// TIA Portal V20 export
DATA_BLOCK "LBP_Axis17"   // DB47
TITLE = Axis-specific signals / Signaux spécifiques à un axe
{ S7_Optimized_Access := 'FALSE' }
AUTHOR : SINUMERIK
FAMILY : SINUMERIK_ONE
VERSION : 6.24
// Interface between user program and axis/spindle, contains signals from/to axis/spindle 17 / Interface entre programme utilisateur et axe/broche, contient des signaux de/vers axe/broche 17
// stored: AutoNumber false, InstanceOfName LBP_typeAxisX, InstanceOfType UDT
"LBP_typeAxisX"
   // VAR RETAIN
   //    A_FD_OR : Byte;
   //    A_DriveEnable : Bool;
   //    A_AckFixedStop : Bool;
   //    A_SensorFixedStop : Bool;
   //    A_ASpDisable : Bool;
   //    A_Follow_upMode : Bool;
   //    A_PosMeas1 : Bool;
   //    A_PosMeas2 : Bool;
   //    A_ORactive : Bool;
   //    A_SWCam : Bool;
   //    A_ContrEnable : Bool;
   //    A_DelDTGSpReset : Bool;
   //    A_Clamp : Bool;
   //    A_RefVal1 : Bool;
   //    A_RefVal2 : Bool;
   //    A_RefVal3 : Bool;
   //    A_RefVal4 : Bool;
   //    A_ExtZO : Bool;
   //    A_EnabTravFixedStop : Bool;
   //    A_FixedFD1 : Bool;
   //    A_FixedFD2 : Bool;
   //    A_FixedFD3 : Bool;
   //    A_FixedFD4 : Bool;
   //    A_VelocSpeedLimit : Bool;
   //    A_PrgtestAxRel : Bool;
   //    A_HW1 : Bool;
   //    A_HW2 : Bool;
   //    A_HW3 : Bool;
   //    A_FDSpStop : Bool;
   //    A_Disable : Bool;
   //    A_RapidTrOR : Bool;
   //    A_Minus : Bool;
   //    A_Plus : Bool;
   //    A_INC1 : Bool;
   //    A_INC10 : Bool;
   //    A_INC100 : Bool;
   //    A_INC1000 : Bool;
   //    A_INC10000 : Bool;
   //    A_INCVar : Bool;
   //    A_ContManTravel : Bool;
   //    f5_7 : Bool;
   //    A_OEMAxis : Byte;
   //    A_InvHWDirOfRot : Bool;
   //    f7_1 : Bool;
   //    f7_2 : Bool;
   //    f7_3 : Bool;
   //    f7_4 : Bool;
   //    f7_5 : Bool;
   //    f7_6 : Bool;
   //    f7_7 : Bool;
   //    A_NCASpChanA : Bool;
   //    A_NCASpChanB : Bool;
   //    A_NCASpChanC : Bool;
   //    A_NCASpChanD : Bool;
   //    A_NCASpStrobe : Bool;
   //    f8_5 : Bool;
   //    f8_6 : Bool;
   //    A_PLCASp : Bool;
   //    A_Para_A : Bool;
   //    A_Para_B : Bool;
   //    A_Para_C : Bool;
   //    A_LockParSetDef : Bool;
   //    f9_4 : Bool;
   //    f9_5 : Bool;
   //    f9_6 : Bool;
   //    f9_7 : Bool;
   //    A_REPOSDelay : Bool;
   //    f10_1 : Bool;
   //    f10_2 : Bool;
   //    f10_3 : Bool;
   //    f10_4 : Bool;
   //    f10_5 : Bool;
   //    f10_6 : Bool;
   //    f10_7 : Bool;
   //    A_StartBrakeTest : Bool;
   //    f11_1 : Bool;
   //    f11_2 : Bool;
   //    f11_3 : Bool;
   //    f11_4 : Bool;
   //    f11_5 : Bool;
   //    f11_6 : Bool;
   //    f11_7 : Bool;
   //    A_HWLimitMinus : Bool;
   //    A_HWLimitPlus : Bool;
   //    A_SWLimit2Minus : Bool;
   //    A_SWLimit2Plus : Bool;
   //    A_ModuloLimitEn : Bool;
   //    f12_5 : Bool;
   //    f12_6 : Bool;
   //    A_DelayRef : Bool;
   //    A_JogFixPPos0 : Bool;
   //    A_JogFixPPos1 : Bool;
   //    A_JogFixPPos2 : Bool;
   //    A_JogToPos : Bool;
   //    f13_4 : Bool;
   //    f13_5 : Bool;
   //    f13_6 : Bool;
   //    f13_7 : Bool;
   //    A_ProgtestSuppress : Bool;
   //    A_ProgtestActivate : Bool;
   //    f14_2 : Bool;
   //    f14_3 : Bool;
   //    f14_4 : Bool;
   //    f14_5 : Bool;
   //    f14_6 : Bool;
   //    f14_7 : Bool;
   //    f15 : Byte;
   //    A_ActGearA : Bool;
   //    A_ActGearB : Bool;
   //    A_ActGearC : Bool;
   //    A_GearChangeOv : Bool;
   //    A_Sp1Syn : Bool;
   //    A_Sp2Syn : Bool;
   //    A_NoMonitorGear : Bool;
   //    A_DeleteS : Bool;
   //    A_FD_ORSp : Bool;
   //    f17_1 : Bool;
   //    f17_2 : Bool;
   //    f17_3 : Bool;
   //    A_Sp1SynP : Bool;
   //    A_Sp2SynP : Bool;
   //    A_M3M4Inv : Bool;
   //    f17_7 : Bool;
   //    f18_0 : Bool;
   //    f18_1 : Bool;
   //    f18_2 : Bool;
   //    f18_3 : Bool;
   //    A_OscilPLC : Bool;
   //    A_OscilSpeed : Bool;
   //    A_SetRotDirectRight : Bool;
   //    A_SetRotDirectLeft : Bool;
   //    A_SpOR : Byte;
   //    f20_0 : Bool;
   //    A_RUEncQuStop : Bool;
   //    f20_2 : Bool;
   //    A_SpeedSetpSmooth : Bool;
   //    f20_4 : Bool;
   //    A_HoldBrakeToOpen : Bool;
   //    f20_6 : Bool;
   //    f20_7 : Bool;
   //    A_ParA : Bool;
   //    A_ParB : Bool;
   //    A_ParC : Bool;
   //    A_MotA : Bool;
   //    A_MotB : Bool;
   //    A_MotOK : Bool;
   //    A_IntegratDisable : Bool;
   //    A_PulseEnable : Bool;
   //    f22_0 : Bool;
   //    f22_1 : Bool;
   //    f22_2 : Bool;
   //    f22_3 : Bool;
   //    f22_4 : Bool;
   //    f22_5 : Bool;
   //    f22_6 : Bool;
   //    f22_7 : Bool;
   //    f23_0 : Bool;
   //    f23_1 : Bool;
   //    f23_2 : Bool;
   //    f23_3 : Bool;
   //    f23_4 : Bool;
   //    f23_5 : Bool;
   //    f23_6 : Bool;
   //    f23_7 : Bool;
   //    f24_0 : Bool;
   //    A_ControlAx : Bool;
   //    f24_2 : Bool;
   //    f24_3 : Bool;
   //    A_TorqComp : Bool;
   //    A_ChangSetpOutAss0 : Bool;
   //    A_ChangSetpOutAss1 : Bool;
   //    A_MS : Bool;
   //    A_DynBComp : Bool;
   //    f25_1 : Bool;
   //    f25_2 : Bool;
   //    f25_3 : Bool;
   //    f25_4 : Bool;
   //    f25_5 : Bool;
   //    f25_6 : Bool;
   //    f25_7 : Bool;
   //    f26_0 : Bool;
   //    f26_1 : Bool;
   //    f26_2 : Bool;
   //    A_CompContr : Bool;
   //    A_FollowAxOv : Bool;
   //    f26_5 : Bool;
   //    f26_6 : Bool;
   //    f26_7 : Bool;
   //    A_DEPMCS : Bool;
   //    A_DEPBCS : Bool;
   //    A_Corr : Bool;
   //    A_HIAxMove : Bool;
   //    A_StopDEPMCS : Bool;
   //    A_StopDEPBCS : Bool;
   //    A_StopCorr : Bool;
   //    A_StopHIAxMove : Bool;
   //    A_OscillAxExtRev : Bool;
   //    A_AxReset : Bool;
   //    A_AxResume : Bool;
   //    A_SetRP : Bool;
   //    A_ChangeRP : Bool;
   //    A_StopRP : Bool;
   //    A_Stop : Bool;
   //    A_PLCAxis : Bool;
   //    f29_0 : Bool;
   //    f29_1 : Bool;
   //    f29_2 : Bool;
   //    f29_3 : Bool;
   //    A_StartGantSynRun : Bool;
   //    A_NoAutoSync : Bool;
   //    f29_6 : Bool;
   //    f29_7 : Bool;
   //    A_StopSpindle : Bool;
   //    A_StartCW : Bool;
   //    A_StartCCW : Bool;
   //    A_AutoGearStep : Bool;
   //    A_PosSpindle : Bool;
   //    f30_5 : Bool;
   //    f30_6 : Bool;
   //    f30_7 : Bool;
   //    f31_0 : Bool;
   //    f31_1 : Bool;
   //    f31_2 : Bool;
   //    f31_3 : Bool;
   //    A_Resynchronize : Bool;
   //    A_DisSync : Bool;
   //    A_Tracksync : Bool;
   //    A_DelSyncRunCorr : Bool;
   //    f32_0 : Bool;
   //    f32_1 : Bool;
   //    f32_2 : Bool;
   //    f32_3 : Bool;
   //    f32_4 : Bool;
   //    f32_5 : Bool;
   //    f32_6 : Bool;
   //    f32_7 : Bool;
   //    f33_0 : Bool;
   //    f33_1 : Bool;
   //    f33_2 : Bool;
   //    f33_3 : Bool;
   //    f33_4 : Bool;
   //    f33_5 : Bool;
   //    f33_6 : Bool;
   //    f33_7 : Bool;
   //    A_SI_SetpLimBit0 : Bool;
   //    A_SI_SetpLimBit1 : Bool;
   //    f34_2 : Bool;
   //    A_ActivateBrakeRampForSs2e : Bool;
   //    f34_4 : Bool;
   //    f34_5 : Bool;
   //    f34_6 : Bool;
   //    f34_7 : Bool;
   //    f35 : Byte;
   //    f36 : Array[36..55] of Byte;
   //    A_FeedDriveCAxEng : Bool;
   //    A_SpSpeedDisp : Bool;
   //    A_SpInsideClamp : Bool;
   //    f56_3 : Bool;
   //    f56_4 : Bool;
   //    f56_5 : Bool;
   //    f56_6 : Bool;
   //    f56_7 : Bool;
   //    f57 : Byte;
   //    f58 : Word;
   //    E_SpNA : Bool;
   //    E_NCU_Link : Bool;
   //    E_EncodFreq1 : Bool;
   //    E_EncodFreq2 : Bool;
   //    E_RefSyn1 : Bool;
   //    E_RefSyn2 : Bool;
   //    E_ExactCoarse : Bool;
   //    E_ExactFine : Bool;
   //    E_TravRequ : Bool;
   //    E_AxialAlarm : Bool;
   //    E_AxisReady : Bool;
   //    E_Follow_upMode : Bool;
   //    E_Stat : Bool;
   //    E_PositContr : Bool;
   //    E_SpeedContr : Bool;
   //    E_CurrentContr : Bool;
   //    E_SWCam : Bool;
   //    E_HWOverlay : Bool;
   //    E_RevFD : Bool;
   //    E_MeasAct : Bool;
   //    E_ActTravFStop : Bool;
   //    E_FixedStop : Bool;
   //    E_ForceFixedStop : Bool;
   //    E_AxContainerRot : Bool;
   //    E_AxReset : Bool;
   //    E_PLCCtrlAx : Bool;
   //    E_AxStop : Bool;
   //    E_AxSpDisable : Bool;
   //    E_StopDEPMCS : Bool;
   //    E_StopDEPBCS : Bool;
   //    E_StopCorr : Bool;
   //    E_StopHIAxMove : Bool;
   //    E_HW1 : Bool;
   //    E_HW2 : Bool;
   //    E_HW3 : Bool;
   //    f64_3 : Bool;
   //    E_TReqMinus : Bool;
   //    E_TReqPlus : Bool;
   //    E_TCMinus : Bool;
   //    E_TCPlus : Bool;
   //    E_INC1 : Bool;
   //    E_INC10 : Bool;
   //    E_INC100 : Bool;
   //    E_INC1000 : Bool;
   //    E_INC10000 : Bool;
   //    E_INCVar : Bool;
   //    E_ContManTravelAct : Bool;
   //    f65_7 : Bool;
   //    E_OEMAxis : Byte;
   //    E_InvHWDirOfRot : Bool;
   //    f67_1 : Bool;
   //    f67_2 : Bool;
   //    f67_3 : Bool;
   //    f67_4 : Bool;
   //    f67_5 : Bool;
   //    f67_6 : Bool;
   //    f67_7 : Bool;
   //    E_NCASpChanA : Bool;
   //    E_NCASpChanB : Bool;
   //    E_NCASpChanC : Bool;
   //    E_NCASpChanD : Bool;
   //    E_PLCType : Bool;
   //    E_ChPoss : Bool;
   //    E_NeutrASp : Bool;
   //    E_PLCASp : Bool;
   //    E_ParS_A : Bool;
   //    E_ParS_B : Bool;
   //    E_ParS_C : Bool;
   //    E_NCUNumLink_3 : Bool;
   //    E_NCUNumLink_4 : Bool;
   //    E_NCUNumLink_5 : Bool;
   //    E_NCUNumLink_6 : Bool;
   //    E_NCUNumLink_7 : Bool;
   //    E_ReposSh : Bool;
   //    E_ReposShValid : Bool;
   //    E_ReposDelayQuit : Bool;
   //    f70_3 : Bool;
   //    f70_4 : Bool;
   //    E_SI_Drv_SICSCC : Bool;
   //    E_SI_Drv_Parameterized : Bool;
   //    f70_7 : Bool;
   //    E_BrakeTest : Bool;
   //    f71_1 : Bool;
   //    f71_2 : Bool;
   //    f71_3 : Bool;
   //    E_POS_RESTORED1 : Bool;
   //    E_POS_RESTORED2 : Bool;
   //    f71_6 : Bool;
   //    E_PLCAxDedic : Bool;
   //    E_MMC_REPOSDelay : Bool;
   //    f72_1 : Bool;
   //    f72_2 : Bool;
   //    f72_3 : Bool;
   //    f72_4 : Bool;
   //    f72_5 : Bool;
   //    f72_6 : Bool;
   //    f72_7 : Bool;
   //    f73 : Byte;
   //    f74_0 : Bool;
   //    f74_1 : Bool;
   //    f74_2 : Bool;
   //    f74_3 : Bool;
   //    E_ModLimEnAct : Bool;
   //    f74_5 : Bool;
   //    f74_6 : Bool;
   //    f74_7 : Bool;
   //    E_JogFixPPos0Act : Bool;
   //    E_JogFixPPos1Act : Bool;
   //    E_JogFixPPos2Act : Bool;
   //    E_JogFixPPos0 : Bool;
   //    E_JogFixPPos1 : Bool;
   //    E_JogFixPPos2 : Bool;
   //    E_JogToPos : Bool;
   //    E_JogPos : Bool;
   //    E_ScratchPulse : Bool;
   //    f76_1 : Bool;
   //    f76_2 : Bool;
   //    f76_3 : Bool;
   //    E_PathAxis : Bool;
   //    E_PosAxis : Bool;
   //    E_IndexAxisPos : Bool;
   //    E_CurvePos : Bool;
   //    E_CollCheckRedSpeed : Bool;
   //    f77_1 : Bool;
   //    f77_2 : Bool;
   //    f77_3 : Bool;
   //    f77_4 : Bool;
   //    f77_5 : Bool;
   //    f77_6 : Bool;
   //    f77_7 : Bool;
   //    E_FPosAxis : Real;
   //    E_SetpGearA : Bool;
   //    E_SetpGearB : Bool;
   //    E_SetpGearC : Bool;
   //    E_GearChange : Bool;
   //    f82_4 : Bool;
   //    f82_5 : Bool;
   //    f82_6 : Bool;
   //    f82_7 : Bool;
   //    E_SpeedLimit : Bool;
   //    E_SetSpeedLimit : Bool;
   //    E_SetSpeedIncreased : Bool;
   //    E_GeoMonit : Bool;
   //    E_SupportAreaViol : Bool;
   //    E_SetRange : Bool;
   //    E_SpeedMonit : Bool;
   //    E_ActRotRight : Bool;
   //    E_ConstCuttSpeed : Bool;
   //    E_SUG : Bool;
   //    E_CLG : Bool;
   //    E_Tapping : Bool;
   //    E_SyncMode : Bool;
   //    E_PosMode : Bool;
   //    E_OscillMode : Bool;
   //    E_ContrMode : Bool;
   //    E_ToolDynLimit : Bool;
   //    f85_1 : Bool;
   //    f85_2 : Bool;
   //    f85_3 : Bool;
   //    f85_4 : Bool;
   //    E_SpInPosition : Bool;
   //    f85_6 : Bool;
   //    f85_7 : Bool;
   //    E_MFunct : Int;
   //    E_SFunct : Real;
   //    f92_0 : Bool;
   //    E_RUEncDisabl : Bool;
   //    f92_2 : Bool;
   //    E_SpeedSetpSmooth : Bool;
   //    E_RLIact : Bool;
   //    E_HoldBrakeOpened : Bool;
   //    f92_6 : Bool;
   //    E_DriveRunEn : Bool;
   //    E_ParA : Bool;
   //    E_ParB : Bool;
   //    E_ParC : Bool;
   //    E_MotA : Bool;
   //    E_MotB : Bool;
   //    E_MotOK : Bool;
   //    E_IntegratDisable : Bool;
   //    E_PulseEnable : Bool;
   //    E_MTempWarn : Bool;
   //    E_HTempWarn : Bool;
   //    E_RUComplete : Bool;
   //    E_MdMdx : Bool;
   //    E_NactNmin : Bool;
   //    E_NactNx : Bool;
   //    E_NactNset : Bool;
   //    E_Message : Bool;
   //    E_UDClessAlThreshold : Bool;
   //    E_DcVoltageAlarmAct : Bool;
   //    E_GeneratorOperationAct : Bool;
   //    E_SpeedBelowMin : Bool;
   //    E_Message2 : Bool;
   //    E_Message3 : Bool;
   //    f95_6 : Bool;
   //    E_I2TLimit : Bool;
   //    f96_0 : Bool;
   //    E_AxisCtrl : Bool;
   //    E_MSFine : Bool;
   //    E_MSCoarse : Bool;
   //    E_MSCompContr : Bool;
   //    E_BitValCtrlOutChang0 : Bool;
   //    E_BitValCtrlOutChang1 : Bool;
   //    E_MS : Bool;
   //    f97 : Byte;
   //    E_SyncronFine : Bool;
   //    E_SyncronCoarse : Bool;
   //    E_ActValCoupling : Bool;
   //    f98_3 : Bool;
   //    E_OverlayMotion : Bool;
   //    E_SWL : Bool;
   //    E_AWL : Bool;
   //    E_EmRetr : Bool;
   //    E_MasterSp : Bool;
   //    E_SlaveSp : Bool;
   //    E_SyncRunCorrDOut : Bool;
   //    E_AxisAccel : Bool;
   //    E_Sync : Bool;
   //    E_MSR : Bool;
   //    E_MAR : Bool;
   //    f99_7 : Bool;
   //    f100_0 : Bool;
   //    f100_1 : Bool;
   //    E_OscillAxExtRev : Bool;
   //    E_StopOscill : Bool;
   //    E_ErrorOscill : Bool;
   //    E_SparkOut : Bool;
   //    E_OscillMotion : Bool;
   //    E_Oscill : Bool;
   //    f101_0 : Bool;
   //    f101_1 : Bool;
   //    E_GantCOLimit : Bool;
   //    E_GantWarn : Bool;
   //    E_SynRunStart : Bool;
   //    E_GantGroupSyn : Bool;
   //    E_GantLeadAxis : Bool;
   //    E_GantAxis : Bool;
   //    E_DynBComp : Bool;
   //    f102_1 : Bool;
   //    f102_2 : Bool;
   //    E_ClampTolerance : Bool;
   //    f102_4 : Bool;
   //    E_PosMeas1 : Bool;
   //    E_PosMeas2 : Bool;
   //    f102_7 : Bool;
   //    E_SyncRunCorrIncl : Bool;
   //    f103_1 : Bool;
   //    f103_2 : Bool;
   //    f103_3 : Bool;
   //    E_Syncron2Fine : Bool;
   //    E_Syncron2Coarse : Bool;
   //    f103_6 : Bool;
   //    f103_7 : Bool;
   //    E_AIAxis : Array[1..31] of Bool;
   //    f108_0 : Bool;
   //    f108_1 : Bool;
   //    f108_2 : Bool;
   //    f108_3 : Bool;
   //    f108_4 : Bool;
   //    f108_5 : Bool;
   //    f108_6 : Bool;
   //    f108_7 : Bool;
   //    f109_0 : Bool;
   //    f109_1 : Bool;
   //    f109_2 : Bool;
   //    f109_3 : Bool;
   //    f109_4 : Bool;
   //    f109_5 : Bool;
   //    f109_6 : Bool;
   //    f109_7 : Bool;
   //    f110_0 : Bool;
   //    f110_1 : Bool;
   //    f110_2 : Bool;
   //    f110_3 : Bool;
   //    f110_4 : Bool;
   //    f110_5 : Bool;
   //    f110_6 : Bool;
   //    f110_7 : Bool;
   //    f111_0 : Bool;
   //    f111_1 : Bool;
   //    f111_2 : Bool;
   //    f111_3 : Bool;
   //    f111_4 : Bool;
   //    f111_5 : Bool;
   //    f111_6 : Bool;
   //    f111_7 : Bool;
   //    f112 : Byte;
   //    f113 : Byte;
   //    f114 : Byte;
   //    f115 : Byte;
   //    f116 : Byte;
   //    f117_0 : Bool;
   //    f117_1 : Bool;
   //    f117_2 : Bool;
   //    f117_3 : Bool;
   //    f117_4 : Bool;
   //    f117_5 : Bool;
   //    f117_6 : Bool;
   //    f117_7 : Bool;
   //    f118 : DWord;
   //    f122 : DWord;
   //    f126 : Word;
   //    E_MMC_ProgtestSuppress : Bool;
   //    E_MMC_ProgtestActivate : Bool;
   //    f128_2 : Bool;
   //    f128_3 : Bool;
   //    f128_4 : Bool;
   //    f128_5 : Bool;
   //    f128_6 : Bool;
   //    f128_7 : Bool;
   //    f129 : Byte;
   //    E_FormatBit0DDS : Bool;
   //    E_FormatBit1DDS : Bool;
   //    E_FormatBit2DDS : Bool;
   //    E_FormatBit3DDS : Bool;
   //    E_FormatBit4DDS : Bool;
   //    f130_5 : Bool;
   //    f130_6 : Bool;
   //    E_MDS_DDS_InterfacesValid : Bool;
   //    f131 : Byte;
   //    E_SensorAv : Bool;
   //    E_S1aMeasARod : Bool;
   //    f132_2 : Bool;
   //    f132_3 : Bool;
   //    E_S4dPistonStopP : Bool;
   //    E_S5dAngleShaft : Bool;
   //    E_S6Temp : Bool;
   //    f132_7 : Bool;
   //    f133 : Byte;
   //    E_ClampingState : Int;
   //    E_AnalogSensor : Int;
   //    f138_0 : Bool;
   //    f138_1 : Bool;
   //    f138_2 : Bool;
   //    f138_3 : Bool;
   //    E_S4PistonStopP : Bool;
   //    E_S5AngleShaft : Bool;
   //    f138_6 : Bool;
   //    f138_7 : Bool;
   //    f139 : Byte;
   //    SCC : Struct
   //       CW1 : Struct
   //          TeststopStart : Bool;
   //          res140_1 : Bool;
   //          res140_2 : Bool;
   //          res140_3 : Bool;
   //          res140_4 : Bool;
   //          CloseBrake : Bool;
   //          res140_6 : Bool;
   //          res140_7 : Bool;
   //          res141 : Byte;
   //       END_STRUCT;
   //       CW3 : Struct
   //          res142 : Byte;
   //          SelectionSBT : Bool;
   //          BT_Start : Bool;
   //          Brake_1_2 : Bool;
   //          DirOfROT : Bool;
   //          Testseq_1_2 : Bool;
   //          BrakeClosed : Bool;
   //          res143_6 : Bool;
   //          res143_7 : Bool;
   //       END_STRUCT;
   //    END_STRUCT;
   //    res144_163 : Array[144..163] of Byte;
   //    SIC : Struct
   //       SW1 : Struct
   //          SLA_Sel : Bool;
   //          SLS_LimBit0_Sel : Bool;
   //          SLS_LimBit1_Sel : Bool;
   //          res164_3 : Bool;
   //          res164_4 : Bool;
   //          res164_5 : Bool;
   //          ESR_Req : Bool;
   //          SF_Message_Act : Bool;
   //          STO_Act : Bool;
   //          SS1_Act : Bool;
   //          SS2_Act : Bool;
   //          SOS_Act : Bool;
   //          SLS_Act : Bool;
   //          SOS_Sel : Bool;
   //          SLS_Sel : Bool;
   //          InternalEvent : Bool;
   //       END_STRUCT;
   //       SW2 : Struct
   //          SDI_P_Sel : Bool;
   //          SDI_N_Sel : Bool;
   //          res166_2 : Bool;
   //          res166_3 : Bool;
   //          TestStopAct : Bool;
   //          TestStopReq : Bool;
   //          res166_6 : Bool;
   //          res166_7 : Bool;
   //          res167_0 : Bool;
   //          res167_1 : Bool;
   //          res167_2 : Bool;
   //          res167_3 : Bool;
   //          SLP_LimBit0_Sel : Bool;
   //          res167_5 : Bool;
   //          res167_6 : Bool;
   //          SLP_Sel : Bool;
   //       END_STRUCT;
   //       V_Limit_B : DInt;
   //       SW3 : Struct
   //          res172_0 : Bool;
   //          res172_1 : Bool;
   //          res172_2 : Bool;
   //          SS2E_ACTIVE : Bool;
   //          SS2ESR : Bool;
   //          res172_5 : Bool;
   //          AcceptSLPAct : Bool;
   //          AcceptTestSel : Bool;
   //          SBT_Sel : Bool;
   //          SetpSettingDrive : Bool;
   //          Brake_1_2 : Bool;
   //          BT_Act : Bool;
   //          BT_OK : Bool;
   //          BT_Finished : Bool;
   //          BrakeReq : Bool;
   //          SignLoadTorque : Bool;
   //       END_STRUCT;
   //    END_STRUCT;
   //    res174_187 : Array[174..187] of Byte;
   //    CW7 : Struct
   //       ReservedBit08 : Bool;
   //       ReservedBit09 : Bool;
   //       ReservedBit10 : Bool;
   //       ReservedBit11 : Bool;
   //       ReservedBit12 : Bool;
   //       ReservedBit13 : Bool;
   //       ReservedBit14 : Bool;
   //       ReservedBit15 : Bool;
   //       A_DisablePowerReduction : Bool;
   //       A_DisableCurrReduction : Bool;
   //       ReservedBit02 : Bool;
   //       ReservedBit03 : Bool;
   //       ReservedBit04 : Bool;
   //       ReservedBit05 : Bool;
   //       ReservedBit06 : Bool;
   //       ReservedBit07 : Bool;
   //    END_STRUCT;
   //    SW7 : Struct
   //       E_EncMaintenanceRequired : Bool;
   //       ReservedBit09 : Bool;
   //       ReservedBit10 : Bool;
   //       ReservedBit11 : Bool;
   //       ReservedBit12 : Bool;
   //       ReservedBit13 : Bool;
   //       ReservedBit14 : Bool;
   //       ReservedBit15 : Bool;
   //       E_TorqueLimited : Bool;
   //       E_CurrReductionActive : Bool;
   //       E_MotorTempModelAlarm : Bool;
   //       E_PolePosIdentPassed : Bool;
   //       ReservedBit04 : Bool;
   //       ReservedBit05 : Bool;
   //       E_AndConditionFulfilled : Bool;
   //       E_OrConditionFulfilled : Bool;
   //    END_STRUCT;
   // END_VAR
BEGIN
END_DATA_BLOCK
